PROGRAM MAIN
VAR_INPUT
	execute : BOOL;
	manualMode : BOOL;
END_VAR
VAR_OUTPUT
	benderLeft : FoldingMachine;
	
	robotLeft, robotRight : Robot;
	
	skidLeft, skidRight : MaterialStorage;
	magazineLeft, magazineRight : MaterialStorage;
	
	wrapper : WrapMachine;
	overhead : STRING;
	
	insertionLeft, insertionRight : ClampInsertion;	
	insertionBottom : TeknicEIP;
	
	innerSuctions, outerSuctions : ARRAY[Surface.TOP_LEFT..Surface.BOTTOM_RIGHT] OF SuctionPad;
END_VAR
VAR
	robotLeftOutputs, robotRightOutputs : ARRAY[1..50] OF INT;
	demoPairCAR : PositionMaterials;
	demoPairCOR : PositionMaterials;
	demoHeight : REAL := 600; //600mm, 60cm
	
	sectionID : SectionEnum := SectionEnum.CARDBOARD_CORNERGUARD;
	
	step : (IDLE, LOAD_CORNERS, LOAD_FLATS, PUSH, RUN_TO_WRAP_POSITION, WRAP_AND_RELEASE, COMPLETE := 1050);
	ready : BOOL;
	
	loadSet : INT;
	loadStepLeft, loadStepRight : INT;
	cornerSetLeft, cornerSetRight : INT;
	
	iWrap : INT;
	wrapPoints : INT;
	wrapRotations : INT;
	
	releaseDelayTimer : TON;
END_VAR
VAR CONSTANT
	releaseDelay : TIME := T#2S;
END_VAR

demoPairCAR.position := 0;
demoPairCAR.top := 'CAR20M';
demoPairCAR.left := 'CAR20S';
demoPairCAR.right := 'CAR20S';
demoPairCAR.bottom := 'CAR28S';
demoPairCAR.wrapRotations := 4;
demoPairCar.wrapPoints := 4;

demoPairCOR.position := 0;
demoPairCOR.topLeft := 'COR48';
demoPairCOR.topRight := 'COR48';
demoPairCOR.bottomLeft := 'COR48';
demoPairCOR.bottomRight := 'COR48';

IF NOT ready THEN
	ready :=
		insertionLeft.homingSequence() AND
		insertionRight.homingSequence() AND
		insertionBottom.homingSequence();
END_IF

CASE step OF
	IDLE:
		IF execute THEN
			execute := FALSE;
			step := LOAD_CORNERS;
		END_IF
	
	LOAD_CORNERS:
		IF load(pair:= demoPairCor) THEN
			IF manualMode AND_THEN NOT execute THEN
				RETURN;
			END_IF
		
			step := LOAD_FLATS;
		END_IF

	LOAD_FLATS:
		IF loadFlats(pair := demoPairCar) THEN
			IF manualMode AND_THEN NOT execute THEN
				RETURN;
			END_IF
		
			step := PUSH;
		END_IF
		
	PUSH:
		insertionBottom.traverse(direction := FALSE);
		IF NOT insertionLeft.alignTarget(demoHeight/2) OR insertionRight.alignTarget(demoHeight/2) THEN
			RETURN;
		END_IF
		
		insertionBottom.traverse(direction := FALSE);
		insertionLeft.press();
		insertionRight.press();
		
		IF insertionBottom.contact AND insertionLeft.contact AND insertionRight.contact THEN
			step := RUN_TO_WRAP_POSITION;
		END_IF
		
	RUN_TO_WRAP_POSITION:
		wrapPoints := MAX(demoPairCAR.wrapPoints, demopairCOR.wrapPoints);
		wrapRotations := MAX(demoPairCAR.wrapRotations, demoPairCOR.wrapRotations);
		
		IF iWrap >= wrapPoints THEN
			step := COMPLETE;
			RETURN;
		END_IF
		
		step := WRAP_AND_RELEASE;
		
	WRAP_AND_RELEASE:
		releaseDelayTimer(IN:= , PT:= releaseDelay, Q=> , ET=> );
		
		IF wrapper.ready OR (NOT wrapper.busy AND NOT wrapper.error) THEN
			wrapper.wrap(wrapRotations);
			releaseDelayTimer.IN := TRUE;
		END_IF
		
		IF releaseDelayTimer.Q THEN
			MEMSET(ADR(innerSuctions), 0, SIZEOF(innerSuctions));
			MEMSET(ADR(outerSuctions), 0, SIZEOF(outerSuctions));
		
			IF NOT insertionLeft.home THEN
				insertionLeft.alignTarget(0);
				insertionLeft.release();
			END_IF
			
			IF NOT insertionRight.home THEN
				insertionRight.alignTarget(0);
				insertionRight.release();
			END_IF
		END_IF		
		
		IF wrapper.done AND insertionLeft.home AND insertionRight.home (*AND insertionBottom.home*) THEN
			releaseDelayTimer.IN := FALSE;
			step := WRAP_AND_RELEASE;
		END_IF
	
	COMPLETE:
		iWrap := wrapPoints := wrapRotations := 0;
		step := IDLE;
		
END_CASE

METHOD changeRobotsEOAT : BOOL
VAR_INPUT
	targetTool : SectionEnum;
END_VAR
(*
IF robotLeft.tool <> sectionID THEN
	MEMSET(ADR(robotLeftOutputs), 0, SIZEOF(robotLeftOutputs));
	robotLeftOutputs[1] := A21.TOOL_CHANGE_CHIPBOARD;
	robotLeft.setParamsAndWait(robotLeftOutputs);
END_IF

IF robotRight.tool <> sectionID THEN
	MEMSET(ADR(robotRightOutputs), 0, SIZEOF(robotRightOutputs));
	robotRightOutputs[1] := A21.TOOL_CHANGE_CHIPBOARD;
	robotRight.setParamsAndWait(robotRightOutputs);
END_IF

changeRobotsEOAT := robotLeft.tool = sectionID AND robotRight.tool = sectionID;
*)
END_METHOD

METHOD hardwareCall : BOOL
benderLeft(enable := TRUE);

robotLeft();
robotRight();

skidLeft();
skidRight();

magazineLeft();
magazineRight();

wrapper();

insertionLeft();
insertionRight();
insertionBottom();
END_METHOD

METHOD PROTECTED leftRobotCornersSequence : BOOL
VAR_IN_OUT
	actingRobot : Robot;
	skid : MaterialStorage;
	loadStep : INT;
END_VAR
VAR_INPUT
	surfaceID : Surface;
	materialID : STRING;
	foldPos0 : INT;
	foldPos1 : INT;
END_VAR
VAR_OUTPUT
	fail : BOOL;
END_VAR
VAR
	slot : INT;
	
	task : INT;
	param0, param1, param2 : INT;
END_VAR
IF materialID = '' THEN
	leftRobotCornersSequence := TRUE;
	RETURN;
END_IF

benderLeft.setFoldingPositions(foldPos0, foldPos1);

CASE loadStep OF
	0: //skid to bender
		IF NOT skid.findSlot(materialID, atSlot=> slot) THEN
			fail := TRUE;
			RETURN;
		END_IF
		
		IF
			actingRobot.setCommandAndWait(
				task:= A22.TRANSFER_TO_BENDER, 
				param1:= slot, 
				param2:= foldPos0, 
				param3:= foldPos1)
		THEN
			loadStep := 10;
		END_IF
		
	10: //bend
		//IF benderLeft.done THEN
			loadStep := 20;
		//END_IF
		
		
	20: //bender to overhead or left insertion
		CASE surfaceID OF
			Surface.TOP_RIGHT, Surface.BOTTOM_RIGHT: //transfer to overhead
				IF overhead <> '' THEN
					RETURN;
				END_IF
				task := A22.TRANSFER_TO_OVERHEAD;
				
			Surface.TOP_LEFT: //load to insertion
				task:= A22.LOAD_BENDER_TO_UPPER_CORNER;
					
			Surface.BOTTOM_LEFT: //load to insertion
				task := A22.LOAD_BENDER_TO_LOWER_CORNER;
				
		END_CASE
		
		IF
			actingRobot.setCommandAndWait(
				task:= task, 
				param1:= param0, 
				param2:= param1, 
				param3:= param1)
		THEN
			 loadStep := COMPLETE;
		END_IF
	
	COMPLETE:
		//turn on suction
		leftRobotCornersSequence := TRUE;
	
END_CASE
END_METHOD

METHOD PROTECTED load : BOOL
VAR_INPUT
	pair : REFERENCE TO PositionMaterials;
END_VAR
IF NOT (robotLeft.operational AND robotRight.operational) THEN
	RETURN;
END_IF

IF NOT (robotLeft.reserve(sectionID) AND robotRight.reserve(sectionID)) THEN //both robots must be reserved first
	RETURN;
END_IF


IF MatchesMaterialType(pair:= pair, materialType:= 'CAR') THEN //is cardboard
	load := loadCornerCardboards(pair:= pair);

ELSIF MatchesMaterialType(pair:= pair, materialType:= 'COR') THEN //is corner guard
	load := loadCornerGuards(pair:= pair);

END_IF


IF load THEN
	robotLeft.release(sectionID);
	robotRight.release(sectionID);
END_IF
END_METHOD

METHOD PROTECTED loadCornerCardboards : BOOL
VAR_INPUT
	pair : REFERENCE TO PositionMaterials;
END_VAR
VAR
	finished : BOOL;
END_VAR
IF cornerSetLeft = 0 THEN //LEFT SIDE
	cornerSetLeft := Surface.TOP_RIGHT;
END_IF

IF
	leftRobotCornersSequence(
		actingRobot:= robotLeft, 
		skid:= skidLeft, 
		surfaceID:= cornerSetLeft,
		loadStep:= loadStepLeft, 
		materialID:= pair.topRight, 
		foldPos0:= pair.topRightFold, 
		foldPos1:= 0, 
		fail=> )
THEN
	CASE cornerSetLeft OF
		Surface.TOP_RIGHT: 
			cornerSetLeft := Surface.TOP_LEFT;
			loadStepLeft := 0;
			
		Surface.TOP_LEFT: 
			cornerSetLeft := Surface.BOTTOM_RIGHT;
			loadStepLeft := 0;
			
		Surface.BOTTOM_RIGHT: 
			cornerSetLeft := Surface.BOTTOM_LEFT;
			loadStepLeft := 0;
			
		Surface.BOTTOM_LEFT: 
			cornerSetLeft := COMPLETE;
			loadStepLeft := COMPLETE;
			
		COMPLETE:
			//
			
	END_CASE
END_IF


IF cornerSetRight = 0 THEN //RIGHT SIDE
	cornerSetRight := Surface.TOP_RIGHT;
END_IF

IF
	rightRobotCornersSequence(
		actingRobot:= robotRight, 
		skid:= skidRight, 
		loadStep:= loadStepRight, 
		materialID:= pair.topRight, 
		surfaceID:= cornerSetRight,
		foldPos1:= pair.topRightFold, 
		foldPos2:= 0, 
		fail=> )
THEN
	CASE cornerSetRight OF
		Surface.TOP_RIGHT: 
			cornerSetRight := Surface.BOTTOM_RIGHT;
			loadStepRight := 0;
			
		Surface.BOTTOM_RIGHT: 
			cornerSetRight := COMPLETE;			
			loadStepRight := COMPLETE;
			
		COMPLETE:
			//
			
	END_CASE
END_IF


IF cornerSetLeft = COMPLETE AND cornerSetRight = COMPLETE THEN
	loadCornerCardboards := TRUE;
	
	loadStepLeft := loadStepRight := 0;
	cornerSetLeft := cornerSetRight := 0;
END_IF
END_METHOD

METHOD PROTECTED loadCornerGuards : BOOL
VAR_INPUT
	pair : REFERENCE TO PositionMaterials;
END_VAR
VAR_OUTPUT
	fail : BOOL;
END_VAR
VAR
	leftFail : BOOL;
	rightFail : BOOL;
END_VAR
CASE loadSet OF
	0: //upper corners
		IF 
			loadGuardSequence(
				actingRobot:= robotLeft, 
				robotOutputs:= robotLeftOutputs, 
				actingStorage:= skidLeft, 
				actingLoadStep:= loadStepLeft, 
				surfaceID:= Surface.TOP_LEFT, 
				material:= pair.topLeft, 
				fail=> leftFail)
			AND
			loadGuardSequence(
				actingRobot:= robotRight, 
				robotOutputs:= robotRightOutputs, 
				actingStorage:= skidRight,
				actingLoadStep:= loadStepRight, 
				surfaceID:= Surface.TOP_RIGHT, 
				material:= pair.topRight, 
				fail=> rightFail)
		THEN
			loadStepLeft := loadStepRight := 0;
			loadSet := 10;
		END_IF
		
	10: //lower corners
		IF 
			loadGuardSequence(
				actingRobot:= robotLeft, 
				robotOutputs:= robotLeftOutputs, 
				actingStorage:= skidLeft, 
				actingLoadStep:= loadStepLeft, 
				surfaceID:= Surface.BOTTOM_LEFT, 
				material:= pair.bottomLeft, 
				fail=> leftFail)
			AND
			loadGuardSequence(
				actingRobot:= robotRight, 
				robotOutputs:= robotRightOutputs, 
				actingStorage:= skidRight,
				actingLoadStep:= loadStepRight, 
				surfaceID:= Surface.BOTTOM_RIGHT, 
				material:= pair.bottomRight, 
				fail=> rightFail)
		THEN
			loadStepLeft := loadStepRight := 0;
			loadSet := COMPLETE;
		END_IF
	
	COMPLETE:
		loadStepLeft := loadStepRight := 0;
		loadSet := 0;
		
		loadCornerGuards := TRUE;
END_CASE

fail := MAX(leftFail, rightFail);
END_METHOD

METHOD PROTECTED loadFlats : BOOL
VAR_INPUT
	pair : REFERENCE TO PositionMaterials;
END_VAR
VAR_OUTPUT
	error : BOOL;
END_VAR
CASE loadSet OF
	0: //top and bottom
		IF 
			loadFlatSequence(
				actingRobot:= robotLeft, 
				robotOutputs:= robotLeftOutputs, 
				actingStorage:= skidLeft, 
				actingLoadStep:= loadStepLeft, 
				surfaceID:= Surface.TOP, 
				material:= pair.top, 
				fail=> )
			AND
			loadFlatSequence(
				actingRobot:= robotRight, 
				robotOutputs:= robotRightOutputs, 
				actingStorage:= skidRight, 
				actingLoadStep:= loadStepRight, 
				surfaceID:= Surface.BOTTOM, 
				material:= pair.bottom, 
				fail=> )
		THEN
			loadStepLeft := loadStepRight := 0;
			loadSet := 10;
		END_IF
		
	10: //sides
		IF 
			loadFlatSequence(
				actingRobot:= robotLeft, 
				robotOutputs:= robotLeftOutputs, 
				actingStorage:= skidLeft, 
				actingLoadStep:= loadStepLeft, 
				surfaceID:= Surface.LEFT, 
				material:= pair.left, 
				fail=> )
			AND
			loadFlatSequence(
				actingRobot:= robotRight, 
				robotOutputs:= robotRightOutputs, 
				actingStorage:= skidRight, 
				actingLoadStep:= loadStepRight, 
				surfaceID:= Surface.RIGHT, 
				material:= pair.right, 
				fail=> )
		THEN
			loadStepLeft := loadStepRight := 0;
			loadSet := COMPLETE;
		END_IF
	
	COMPLETE:
		loadStepLeft := loadStepRight := 0;
		loadSet := 0;
		
		loadFlats := TRUE;
END_CASE
END_METHOD

METHOD loadFlatSequence : BOOL
VAR_IN_OUT
	actingRobot : Robot;
	robotOutputs : ARRAY[1..50] OF INT;
	actingStorage : MaterialStorage;
	actingLoadStep : INT;
END_VAR
VAR_INPUT
	surfaceID : Surface;
	material : STRING;
END_VAR
VAR_OUTPUT
	fail : BOOL;
END_VAR
VAR
	slot : INT;
END_VAR
IF material = '' THEN
	loadFlatSequence := TRUE;
	RETURN;
END_IF

CASE actingLoadStep OF
	0:
		IF NOT actingStorage.findSlot(materialID := material, atSlot => slot) THEN
			fail := TRUE;
			RETURN;
		END_IF
		
		MEMSET(ADR(robotOutputs), 0, SIZEOF(robotOutputs));
		CASE surfaceID OF
			Surface.TOP: 					robotOutputs[1] := A22.LOAD_CARDBOARD_TOP;
			Surface.LEFT, Surface.RIGHT: 	robotOutputs[1] := A22.LOAD_CARDBOARD_SIDE;
			Surface.BOTTOM: 				robotOutputs[1] := A22.LOAD_CARDBOARD_BOTTOM;
		END_CASE
		robotOutputs[2] := slot;
		
		IF actingRobot.setParamsAndWait(robotOutputs) THEN
			actingLoadStep := COMPLETE;
		END_IF
		
	COMPLETE:
		loadFlatSequence := TRUE;
	
END_CASE
END_METHOD

METHOD loadGuardSequence : BOOL
VAR_IN_OUT
	actingRobot : Robot;
	robotOutputs : ARRAY[1..50] OF INT;
	actingStorage : MaterialStorage;
	actingLoadStep : INT;
END_VAR
VAR_INPUT
	surfaceID : Surface;
	material : STRING;
END_VAR
VAR_OUTPUT
	fail : BOOL;
END_VAR
VAR
	slot : INT;
END_VAR
IF material = '' THEN
	loadGuardSequence := TRUE;
	RETURN;
END_IF

CASE actingLoadStep OF
	0:
		IF NOT actingStorage.findSlot(materialID := material, atSlot => slot) THEN //load from staging table
			fail := TRUE;
			RETURN;
		END_IF
		
		MEMSET(ADR(robotOutputs), 0, SIZEOF(robotOutputs));
		CASE surfaceID OF
			Surface.TOP_LEFT, Surface.TOP_RIGHT: 		robotOutputs[1] := A22.LOAD_CORNER_GUARD_UPPER;
			Surface.BOTTOM_LEFT, Surface.BOTTOM_RIGHT:	robotOutputs[1] := A22.LOAD_CORNER_GUARD_LOWER;
		END_CASE
		robotOutputs[2] := slot;
		
		IF actingRobot.setParamsAndWait(robotOutputs) THEN
			actingLoadStep := COMPLETE;
		END_IF
		
	COMPLETE:
		outerSuctions[surfaceID].enable := TRUE;
		loadGuardSequence := TRUE;
END_CASE
END_METHOD

METHOD PROTECTED rightRobotCornersSequence : BOOL
VAR_IN_OUT
	actingRobot : Robot;
	skid : MaterialStorage;
	loadStep : INT;
END_VAR
VAR_INPUT
	surfaceID : Surface;
	materialID : STRING;
	foldPos1 : INT;
	foldPos2 : INT;
END_VAR
VAR_OUTPUT
	fail : BOOL;
END_VAR
VAR
	slot : INT;
	
	task : INT;
	param0, param1, param2 : INT;
END_VAR
IF materialID = '' THEN
	rightRobotCornersSequence := TRUE;
	RETURN;
END_IF

CASE loadStep OF
	0: //overhead to insertion
		IF overhead = '' THEN
			RETURN;
		END_IF
		
		CASE surfaceID OF
			Surface.TOP_RIGHT:
				task := A22.LOAD_OVERHEAD_TO_UPPER_CORNER;
				
			Surface.BOTTOM_RIGHT:
				task := A22.LOAD_OVERHEAD_TO_LOWER_CORNER;
				
		END_CASE
		
		IF
			actingRobot.setCommandAndWait(
				task:= task, 
				param1:= slot, 
				param2:= foldPos1, 
				param3:= foldPos2)
		THEN
			loadStep := COMPLETE;
		END_IF
	
	COMPLETE:
		//turn on suction
		rightRobotCornersSequence := TRUE;
	
END_CASE
END_METHOD

END_PROGRAM

(* stored: Version 1.1.0.1, ProductVersion 3.1.4024.11
   POU MAIN: Id {bb23f57b-bfaa-4807-862f-695fb779bd1d}, SpecialFunc None
   Folder Cardboard (Corner): Id {75e45005-57b6-45af-977a-1cc75cf19289}
   Folder Cardboard (Flat): Id {69bbbb84-f428-46bc-8482-36bd2217074a}
   Folder Corner Guards: Id {6138b1d4-74c6-4a8f-864e-6193654c592a}
   Method changeRobotsEOAT: Id {71a414a6-260d-4ed7-9b91-4169239414f1}
   Method hardwareCall: Id {ae27e4e1-f18c-46c6-a88d-05763e2b1498}
   Method leftRobotCornersSequence: Id {08bffef9-e349-4b7d-9ae3-92f5a7d8876a}
   Method load: Id {a681c93d-e590-4020-9185-d7ae010cf638}
   Method loadCornerCardboards: Id {fc6e26f1-7233-42c4-a94a-66d2e256266a}
   Method loadCornerGuards: Id {73216583-3bb4-409e-896a-e96f29db7009}
   Method loadFlats: Id {b9a93d4c-938b-4af6-a5a3-5141d50c48d4}
   Method loadFlatSequence: Id {e9b25173-0158-437d-9616-4153dd5d3500}
   Method loadGuardSequence: Id {6d84fe42-26e5-4a1f-b580-8cefdfabe586}
   Method rightRobotCornersSequence: Id {879cd7f3-c4e8-4979-a4c5-8a1bacb14790} *)
